; ----- Contour 7 -----
PTP {X 40.51, Y 258.85, Z 10.00, A 0, B 0, C 0}
LIN {X 40.51, Y 258.85, Z 0.00, A 0, B 0, C 0}
LIN {X 40.30, Y 258.74, Z 0.00, A 0, B 0, C 0} C_DIS
LIN {X 40.09, Y 258.64, Z 0.00, A 0, B 0, C 0} C_DIS
LIN {X 39.88, Y 258.57, Z 0.00, A 0, B 0, C 0} C_DIS
LIN {X 39.67, Y 258.50, Z 0.00, A 0, B 0, C 0} C_DIS
LIN {X 39.46, Y 258.46, Z 0.00, A 0, B 0, C 0} C_DIS
LIN {X 39.25, Y 258.42, Z 0.00, A 0, B 0, C 0} C_DIS
LIN {X 39.03, Y 258.40, Z 0.00, A 0, B 0, C 0} C_DIS
LIN {X 38.81, Y 258.38, Z 0.00, A 0, B 0, C 0} C_DIS
LIN {X 38.60, Y 258.38, Z 0.00, A 0, B 0, C 0} C_DIS
LIN {X 38.38, Y 258.38, Z 0.00, A 0, B 0, C 0} C_DIS
LIN {X 38.16, Y 258.38, Z 0.00, A 0, B 0, C 0} C_DIS
LIN {X 37.94, Y 258.39, Z 0.00, A 0, B 0, C 0} C_DIS
LIN {X 37.72, Y 258.39, Z 0.00, A 0, B 0, C 0} C_DIS
LIN {X 37.51, Y 258.40, Z 0.00, A 0, B 0, C 0} C_DIS
LIN {X 37.29, Y 258.41, Z 0.00, A 0, B 0, C 0} C_DIS
LIN {X 37.07, Y 258.41, Z 0.00, A 0, B 0, C 0} C_DIS
LIN {X 36.85, Y 258.42, Z 0.00, A 0, B 0, C 0} C_DIS
LIN {X 36.63, Y 258.42, Z 0.00, A 0, B 0, C 0} C_DIS
LIN {X 36.42, Y 258.42, Z 0.00, A 0, B 0, C 0} C_DIS
LIN {X 36.20, Y 258.42, Z 0.00, A 0, B 0, C 0} C_DIS
LIN {X 35.98, Y 258.42, Z 0.00, A 0, B 0, C 0} C_DIS
LIN {X 35.76, Y 258.42, Z 0.00, A 0, B 0, C 0} C_DIS
LIN {X 35.55, Y 258.42, Z 0.00, A 0, B 0, C 0} C_DIS
LIN {X 35.33, Y 258.42, Z 0.00, A 0, B 0, C 0} C_DIS
LIN {X 35.11, Y 258.41, Z 0.00, A 0, B 0, C 0} C_DIS
LIN {X 34.90, Y 258.41, Z 0.00, A 0, B 0, C 0} C_DIS
LIN {X 34.68, Y 258.41, Z 0.00, A 0, B 0, C 0} C_DIS
LIN {X 34.46, Y 258.41, Z 0.00, A 0, B 0, C 0} C_DIS
LIN {X 34.24, Y 258.41, Z 0.00, A 0, B 0, C 0} C_DIS
LIN {X 34.03, Y 258.40, Z 0.00, A 0, B 0, C 0} C_DIS
LIN {X 33.81, Y 258.40, Z 0.00, A 0, B 0, C 0} C_DIS
LIN {X 33.59, Y 258.40, Z 0.00, A 0, B 0, C 0} C_DIS
LIN {X 33.37, Y 258.40, Z 0.00, A 0, B 0, C 0} C_DIS
LIN {X 33.16, Y 258.40, Z 0.00, A 0, B 0, C 0} C_DIS
LIN {X 32.94, Y 258.40, Z 0.00, A 0, B 0, C 0} C_DIS
LIN {X 32.72, Y 258.40, Z 0.00, A 0, B 0, C 0} C_DIS
LIN {X 32.51, Y 258.40, Z 0.00, A 0, B 0, C 0} C_DIS
LIN {X 32.29, Y 258.40, Z 0.00, A 0, B 0, C 0} C_DIS
LIN {X 32.07, Y 258.40, Z 0.00, A 0, B 0, C 0} C_DIS
LIN {X 31.85, Y 258.40, Z 0.00, A 0, B 0, C 0} C_DIS
LIN {X 31.64, Y 258.40, Z 0.00, A 0, B 0, C 0} C_DIS
LIN {X 31.42, Y 258.40, Z 0.00, A 0, B 0, C 0} C_DIS
LIN {X 31.20, Y 258.40, Z 0.00, A 0, B 0, C 0} C_DIS
LIN {X 30.98, Y 258.40, Z 0.00, A 0, B 0, C 0} C_DIS
LIN {X 30.77, Y 258.40, Z 0.00, A 0, B 0, C 0} C_DIS
LIN {X 30.55, Y 258.40, Z 0.00, A 0, B 0, C 0} C_DIS
LIN {X 30.33, Y 258.40, Z 0.00, A 0, B 0, C 0} C_DIS
LIN {X 30.11, Y 258.41, Z 0.00, A 0, B 0, C 0} C_DIS
LIN {X 29.90, Y 258.41, Z 0.00, A 0, B 0, C 0} C_DIS
LIN {X 29.68, Y 258.41, Z 0.00, A 0, B 0, C 0} C_DIS
LIN {X 29.46, Y 258.41, Z 0.00, A 0, B 0, C 0} C_DIS
LIN {X 29.25, Y 258.41, Z 0.00, A 0, B 0, C 0} C_DIS
LIN {X 29.03, Y 258.41, Z 0.00, A 0, B 0, C 0} C_DIS
LIN {X 28.81, Y 258.41, Z 0.00, A 0, B 0, C 0} C_DIS
LIN {X 28.59, Y 258.41, Z 0.00, A 0, B 0, C 0} C_DIS
LIN {X 28.38, Y 258.41, Z 0.00, A 0, B 0, C 0} C_DIS
LIN {X 28.16, Y 258.41, Z 0.00, A 0, B 0, C 0} C_DIS
LIN {X 27.94, Y 258.41, Z 0.00, A 0, B 0, C 0} C_DIS
LIN {X 27.72, Y 258.41, Z 0.00, A 0, B 0, C 0} C_DIS
LIN {X 27.51, Y 258.41, Z 0.00, A 0, B 0, C 0} C_DIS
LIN {X 27.29, Y 258.41, Z 0.00, A 0, B 0, C 0} C_DIS
LIN {X 27.07, Y 258.41, Z 0.00, A 0, B 0, C 0} C_DIS
LIN {X 26.85, Y 258.41, Z 0.00, A 0, B 0, C 0} C_DIS
LIN {X 26.64, Y 258.41, Z 0.00, A 0, B 0, C 0} C_DIS
LIN {X 26.42, Y 258.41, Z 0.00, A 0, B 0, C 0} C_DIS
LIN {X 26.20, Y 258.41, Z 0.00, A 0, B 0, C 0} C_DIS
LIN {X 25.98, Y 258.41, Z 0.00, A 0, B 0, C 0} C_DIS
LIN {X 25.77, Y 258.41, Z 0.00, A 0, B 0, C 0} C_DIS
LIN {X 25.55, Y 258.41, Z 0.00, A 0, B 0, C 0} C_DIS
LIN {X 25.33, Y 258.41, Z 0.00, A 0, B 0, C 0} C_DIS
LIN {X 25.11, Y 258.41, Z 0.00, A 0, B 0, C 0} C_DIS
LIN {X 24.90, Y 258.41, Z 0.00, A 0, B 0, C 0} C_DIS
LIN {X 24.68, Y 258.41, Z 0.00, A 0, B 0, C 0} C_DIS
LIN {X 24.46, Y 258.41, Z 0.00, A 0, B 0, C 0} C_DIS
LIN {X 24.24, Y 258.41, Z 0.00, A 0, B 0, C 0} C_DIS
LIN {X 24.03, Y 258.41, Z 0.00, A 0, B 0, C 0} C_DIS
LIN {X 23.81, Y 258.41, Z 0.00, A 0, B 0, C 0} C_DIS
LIN {X 23.59, Y 258.41, Z 0.00, A 0, B 0, C 0} C_DIS
LIN {X 23.37, Y 258.41, Z 0.00, A 0, B 0, C 0} C_DIS
LIN {X 23.16, Y 258.41, Z 0.00, A 0, B 0, C 0} C_DIS
LIN {X 22.94, Y 258.41, Z 0.00, A 0, B 0, C 0} C_DIS
LIN {X 22.72, Y 258.41, Z 0.00, A 0, B 0, C 0} C_DIS
LIN {X 22.51, Y 258.41, Z 0.00, A 0, B 0, C 0} C_DIS
LIN {X 22.29, Y 258.41, Z 0.00, A 0, B 0, C 0} C_DIS
LIN {X 22.07, Y 258.41, Z 0.00, A 0, B 0, C 0} C_DIS
LIN {X 21.85, Y 258.40, Z 0.00, A 0, B 0, C 0} C_DIS
LIN {X 21.64, Y 258.40, Z 0.00, A 0, B 0, C 0} C_DIS
LIN {X 21.42, Y 258.40, Z 0.00, A 0, B 0, C 0} C_DIS
LIN {X 21.20, Y 258.40, Z 0.00, A 0, B 0, C 0} C_DIS
LIN {X 20.98, Y 258.40, Z 0.00, A 0, B 0, C 0} C_DIS
LIN {X 20.77, Y 258.40, Z 0.00, A 0, B 0, C 0} C_DIS
LIN {X 20.55, Y 258.40, Z 0.00, A 0, B 0, C 0} C_DIS
LIN {X 20.33, Y 258.40, Z 0.00, A 0, B 0, C 0} C_DIS
LIN {X 20.11, Y 258.40, Z 0.00, A 0, B 0, C 0} C_DIS
LIN {X 19.90, Y 258.40, Z 0.00, A 0, B 0, C 0} C_DIS
LIN {X 19.68, Y 258.40, Z 0.00, A 0, B 0, C 0} C_DIS
LIN {X 19.46, Y 258.40, Z 0.00, A 0, B 0, C 0} C_DIS
LIN {X 19.24, Y 258.40, Z 0.00, A 0, B 0, C 0} C_DIS
LIN {X 19.03, Y 258.40, Z 0.00, A 0, B 0, C 0} C_DIS
LIN {X 18.81, Y 258.40, Z 0.00, A 0, B 0, C 0} C_DIS
LIN {X 18.59, Y 258.40, Z 0.00, A 0, B 0, C 0} C_DIS
LIN {X 18.37, Y 258.40, Z 0.00, A 0, B 0, C 0} C_DIS
LIN {X 18.16, Y 258.40, Z 0.00, A 0, B 0, C 0} C_DIS
LIN {X 17.94, Y 258.40, Z 0.00, A 0, B 0, C 0} C_DIS
LIN {X 17.72, Y 258.40, Z 0.00, A 0, B 0, C 0} C_DIS
LIN {X 17.50, Y 258.40, Z 0.00, A 0, B 0, C 0} C_DIS
LIN {X 17.29, Y 258.40, Z 0.00, A 0, B 0, C 0} C_DIS
LIN {X 17.07, Y 258.40, Z 0.00, A 0, B 0, C 0} C_DIS
LIN {X 16.85, Y 258.40, Z 0.00, A 0, B 0, C 0} C_DIS
LIN {X 16.64, Y 258.40, Z 0.00, A 0, B 0, C 0} C_DIS
LIN {X 16.42, Y 258.40, Z 0.00, A 0, B 0, C 0} C_DIS
LIN {X 16.20, Y 258.40, Z 0.00, A 0, B 0, C 0} C_DIS
LIN {X 15.98, Y 258.40, Z 0.00, A 0, B 0, C 0} C_DIS
LIN {X 15.77, Y 258.40, Z 0.00, A 0, B 0, C 0} C_DIS
LIN {X 15.55, Y 258.40, Z 0.00, A 0, B 0, C 0} C_DIS
LIN {X 15.33, Y 258.40, Z 0.00, A 0, B 0, C 0} C_DIS
LIN {X 15.11, Y 258.40, Z 0.00, A 0, B 0, C 0} C_DIS
LIN {X 14.90, Y 258.40, Z 0.00, A 0, B 0, C 0} C_DIS
LIN {X 14.68, Y 258.40, Z 0.00, A 0, B 0, C 0} C_DIS
LIN {X 14.46, Y 258.41, Z 0.00, A 0, B 0, C 0} C_DIS
LIN {X 14.24, Y 258.41, Z 0.00, A 0, B 0, C 0} C_DIS
LIN {X 14.03, Y 258.41, Z 0.00, A 0, B 0, C 0} C_DIS
LIN {X 13.81, Y 258.41, Z 0.00, A 0, B 0, C 0} C_DIS
LIN {X 13.59, Y 258.41, Z 0.00, A 0, B 0, C 0} C_DIS
LIN {X 13.38, Y 258.41, Z 0.00, A 0, B 0, C 0} C_DIS
LIN {X 13.16, Y 258.41, Z 0.00, A 0, B 0, C 0} C_DIS
LIN {X 12.94, Y 258.41, Z 0.00, A 0, B 0, C 0} C_DIS
LIN {X 12.72, Y 258.41, Z 0.00, A 0, B 0, C 0} C_DIS
LIN {X 12.51, Y 258.41, Z 0.00, A 0, B 0, C 0} C_DIS
LIN {X 12.29, Y 258.41, Z 0.00, A 0, B 0, C 0} C_DIS
LIN {X 12.07, Y 258.42, Z 0.00, A 0, B 0, C 0} C_DIS
LIN {X 11.85, Y 258.42, Z 0.00, A 0, B 0, C 0} C_DIS
LIN {X 11.64, Y 258.42, Z 0.00, A 0, B 0, C 0} C_DIS
LIN {X 11.42, Y 258.42, Z 0.00, A 0, B 0, C 0} C_DIS
LIN {X 11.20, Y 258.42, Z 0.00, A 0, B 0, C 0} C_DIS
LIN {X 10.98, Y 258.42, Z 0.00, A 0, B 0, C 0} C_DIS
LIN {X 10.77, Y 258.42, Z 0.00, A 0, B 0, C 0} C_DIS
LIN {X 10.55, Y 258.42, Z 0.00, A 0, B 0, C 0} C_DIS
LIN {X 10.33, Y 258.42, Z 0.00, A 0, B 0, C 0} C_DIS
LIN {X 10.12, Y 258.42, Z 0.00, A 0, B 0, C 0} C_DIS
LIN {X 9.90, Y 258.42, Z 0.00, A 0, B 0, C 0} C_DIS
LIN {X 9.68, Y 258.42, Z 0.00, A 0, B 0, C 0} C_DIS
LIN {X 9.46, Y 258.42, Z 0.00, A 0, B 0, C 0} C_DIS
LIN {X 9.25, Y 258.42, Z 0.00, A 0, B 0, C 0} C_DIS
LIN {X 9.03, Y 258.42, Z 0.00, A 0, B 0, C 0} C_DIS
LIN {X 8.81, Y 258.42, Z 0.00, A 0, B 0, C 0} C_DIS
LIN {X 8.59, Y 258.42, Z 0.00, A 0, B 0, C 0} C_DIS
LIN {X 8.38, Y 258.42, Z 0.00, A 0, B 0, C 0} C_DIS
LIN {X 8.16, Y 258.42, Z 0.00, A 0, B 0, C 0} C_DIS
LIN {X 7.94, Y 258.42, Z 0.00, A 0, B 0, C 0} C_DIS
LIN {X 7.72, Y 258.42, Z 0.00, A 0, B 0, C 0} C_DIS
LIN {X 7.51, Y 258.42, Z 0.00, A 0, B 0, C 0} C_DIS
LIN {X 7.29, Y 258.42, Z 0.00, A 0, B 0, C 0} C_DIS
LIN {X 7.07, Y 258.41, Z 0.00, A 0, B 0, C 0} C_DIS
LIN {X 6.85, Y 258.41, Z 0.00, A 0, B 0, C 0} C_DIS
LIN {X 6.63, Y 258.41, Z 0.00, A 0, B 0, C 0} C_DIS
LIN {X 6.42, Y 258.41, Z 0.00, A 0, B 0, C 0} C_DIS
LIN {X 6.20, Y 258.41, Z 0.00, A 0, B 0, C 0} C_DIS
LIN {X 5.98, Y 258.40, Z 0.00, A 0, B 0, C 0} C_DIS
LIN {X 5.76, Y 258.40, Z 0.00, A 0, B 0, C 0} C_DIS
LIN {X 5.55, Y 258.40, Z 0.00, A 0, B 0, C 0} C_DIS
LIN {X 5.33, Y 258.40, Z 0.00, A 0, B 0, C 0} C_DIS
LIN {X 5.11, Y 258.39, Z 0.00, A 0, B 0, C 0} C_DIS
LIN {X 4.89, Y 258.39, Z 0.00, A 0, B 0, C 0} C_DIS
LIN {X 4.68, Y 258.39, Z 0.00, A 0, B 0, C 0} C_DIS
LIN {X 4.46, Y 258.38, Z 0.00, A 0, B 0, C 0} C_DIS
LIN {X 4.24, Y 258.38, Z 0.00, A 0, B 0, C 0} C_DIS
LIN {X 4.02, Y 258.38, Z 0.00, A 0, B 0, C 0} C_DIS
LIN {X 3.80, Y 258.37, Z 0.00, A 0, B 0, C 0} C_DIS
LIN {X 3.59, Y 258.36, Z 0.00, A 0, B 0, C 0} C_DIS
LIN {X 3.37, Y 258.35, Z 0.00, A 0, B 0, C 0} C_DIS
LIN {X 3.16, Y 258.32, Z 0.00, A 0, B 0, C 0} C_DIS
LIN {X 2.94, Y 258.29, Z 0.00, A 0, B 0, C 0} C_DIS
LIN {X 2.74, Y 258.24, Z 0.00, A 0, B 0, C 0} C_DIS
LIN {X 2.53, Y 258.18, Z 0.00, A 0, B 0, C 0} C_DIS
LIN {X 2.33, Y 258.09, Z 0.00, A 0, B 0, C 0} C_DIS
LIN {X 2.13, Y 257.99, Z 0.00, A 0, B 0, C 0} C_DIS
LIN {X 1.94, Y 257.86, Z 0.00, A 0, B 0, C 0} C_DIS
LIN {X 1.75, Y 257.71, Z 0.00, A 0, B 0, C 0} C_DIS
LIN {X 1.57, Y 257.52, Z 0.00, A 0, B 0, C 0} C_DIS
LIN {X 1.40, Y 257.31, Z 0.00, A 0, B 0, C 0} C_DIS
LIN {X 1.23, Y 257.08, Z 0.00, A 0, B 0, C 0} C_DIS
LIN {X 1.07, Y 256.83, Z 0.00, A 0, B 0, C 0} C_DIS
LIN {X 0.92, Y 256.56, Z 0.00, A 0, B 0, C 0} C_DIS
LIN {X 0.78, Y 256.30, Z 0.00, A 0, B 0, C 0} C_DIS
LIN {X 0.65, Y 256.03, Z 0.00, A 0, B 0, C 0} C_DIS
LIN {X 0.53, Y 255.76, Z 0.00, A 0, B 0, C 0} C_DIS
LIN {X 0.42, Y 255.48, Z 0.00, A 0, B 0, C 0} C_DIS
LIN {X 0.32, Y 255.20, Z 0.00, A 0, B 0, C 0} C_DIS
LIN {X 0.23, Y 254.91, Z 0.00, A 0, B 0, C 0} C_DIS
LIN {X 0.16, Y 254.61, Z 0.00, A 0, B 0, C 0} C_DIS
LIN {X 0.09, Y 254.30, Z 0.00, A 0, B 0, C 0} C_DIS
LIN {X 0.04, Y 253.99, Z 0.00, A 0, B 0, C 0} C_DIS
LIN {X -0.01, Y 253.66, Z 0.00, A 0, B 0, C 0} C_DIS
LIN {X -0.04, Y 253.34, Z 0.00, A 0, B 0, C 0} C_DIS
LIN {X -0.06, Y 253.01, Z 0.00, A 0, B 0, C 0} C_DIS
LIN {X -0.07, Y 252.68, Z 0.00, A 0, B 0, C 0} C_DIS
LIN {X -0.06, Y 252.35, Z 0.00, A 0, B 0, C 0} C_DIS
LIN {X -0.05, Y 252.02, Z 0.00, A 0, B 0, C 0} C_DIS
LIN {X -0.03, Y 251.70, Z 0.00, A 0, B 0, C 0} C_DIS
LIN {X 0.01, Y 251.37, Z 0.00, A 0, B 0, C 0} C_DIS
LIN {X 0.06, Y 251.06, Z 0.00, A 0, B 0, C 0} C_DIS
LIN {X 0.12, Y 250.74, Z 0.00, A 0, B 0, C 0} C_DIS
LIN {X 0.19, Y 250.44, Z 0.00, A 0, B 0, C 0} C_DIS
LIN {X 0.27, Y 250.14, Z 0.00, A 0, B 0, C 0} C_DIS
LIN {X 0.36, Y 249.85, Z 0.00, A 0, B 0, C 0} C_DIS
LIN {X 0.46, Y 249.56, Z 0.00, A 0, B 0, C 0} C_DIS
LIN {X 0.57, Y 249.29, Z 0.00, A 0, B 0, C 0} C_DIS
LIN {X 0.69, Y 249.02, Z 0.00, A 0, B 0, C 0} C_DIS
LIN {X 0.83, Y 248.76, Z 0.00, A 0, B 0, C 0} C_DIS
LIN {X 0.97, Y 248.51, Z 0.00, A 0, B 0, C 0} C_DIS
LIN {X 1.12, Y 248.27, Z 0.00, A 0, B 0, C 0} C_DIS
LIN {X 1.28, Y 248.04, Z 0.00, A 0, B 0, C 0} C_DIS
LIN {X 1.45, Y 247.82, Z 0.00, A 0, B 0, C 0} C_DIS
LIN {X 1.62, Y 247.62, Z 0.00, A 0, B 0, C 0} C_DIS
LIN {X 1.81, Y 247.43, Z 0.00, A 0, B 0, C 0} C_DIS
LIN {X 1.99, Y 247.27, Z 0.00, A 0, B 0, C 0} C_DIS
LIN {X 2.19, Y 247.13, Z 0.00, A 0, B 0, C 0} C_DIS
LIN {X 2.39, Y 247.02, Z 0.00, A 0, B 0, C 0} C_DIS
LIN {X 2.59, Y 246.93, Z 0.00, A 0, B 0, C 0} C_DIS
LIN {X 2.80, Y 246.87, Z 0.00, A 0, B 0, C 0} C_DIS
LIN {X 3.01, Y 246.82, Z 0.00, A 0, B 0, C 0} C_DIS
LIN {X 3.23, Y 246.79, Z 0.00, A 0, B 0, C 0} C_DIS
LIN {X 3.44, Y 246.77, Z 0.00, A 0, B 0, C 0} C_DIS
LIN {X 3.66, Y 246.75, Z 0.00, A 0, B 0, C 0} C_DIS
LIN {X 3.88, Y 246.74, Z 0.00, A 0, B 0, C 0} C_DIS
LIN {X 4.09, Y 246.73, Z 0.00, A 0, B 0, C 0} C_DIS
LIN {X 4.31, Y 246.72, Z 0.00, A 0, B 0, C 0} C_DIS
LIN {X 4.53, Y 246.72, Z 0.00, A 0, B 0, C 0} C_DIS
LIN {X 4.74, Y 246.71, Z 0.00, A 0, B 0, C 0} C_DIS
LIN {X 4.96, Y 246.71, Z 0.00, A 0, B 0, C 0} C_DIS
LIN {X 5.18, Y 246.71, Z 0.00, A 0, B 0, C 0} C_DIS
LIN {X 5.40, Y 246.71, Z 0.00, A 0, B 0, C 0} C_DIS
LIN {X 5.62, Y 246.71, Z 0.00, A 0, B 0, C 0} C_DIS
LIN {X 5.83, Y 246.72, Z 0.00, A 0, B 0, C 0} C_DIS
LIN {X 6.05, Y 246.72, Z 0.00, A 0, B 0, C 0} C_DIS
LIN {X 6.27, Y 246.72, Z 0.00, A 0, B 0, C 0} C_DIS
LIN {X 6.49, Y 246.73, Z 0.00, A 0, B 0, C 0} C_DIS
LIN {X 6.70, Y 246.73, Z 0.00, A 0, B 0, C 0} C_DIS
LIN {X 6.92, Y 246.73, Z 0.00, A 0, B 0, C 0} C_DIS
LIN {X 7.14, Y 246.74, Z 0.00, A 0, B 0, C 0} C_DIS
LIN {X 7.36, Y 246.74, Z 0.00, A 0, B 0, C 0} C_DIS
LIN {X 7.58, Y 246.74, Z 0.00, A 0, B 0, C 0} C_DIS
LIN {X 7.79, Y 246.74, Z 0.00, A 0, B 0, C 0} C_DIS
LIN {X 8.01, Y 246.74, Z 0.00, A 0, B 0, C 0} C_DIS
LIN {X 8.23, Y 246.75, Z 0.00, A 0, B 0, C 0} C_DIS
LIN {X 8.45, Y 246.75, Z 0.00, A 0, B 0, C 0} C_DIS
LIN {X 8.66, Y 246.75, Z 0.00, A 0, B 0, C 0} C_DIS
LIN {X 8.88, Y 246.75, Z 0.00, A 0, B 0, C 0} C_DIS
LIN {X 9.10, Y 246.75, Z 0.00, A 0, B 0, C 0} C_DIS
LIN {X 9.31, Y 246.75, Z 0.00, A 0, B 0, C 0} C_DIS
LIN {X 9.53, Y 246.75, Z 0.00, A 0, B 0, C 0} C_DIS
LIN {X 9.75, Y 246.75, Z 0.00, A 0, B 0, C 0} C_DIS
LIN {X 9.97, Y 246.75, Z 0.00, A 0, B 0, C 0} C_DIS
LIN {X 10.18, Y 246.75, Z 0.00, A 0, B 0, C 0} C_DIS
LIN {X 10.40, Y 246.75, Z 0.00, A 0, B 0, C 0} C_DIS
LIN {X 10.62, Y 246.75, Z 0.00, A 0, B 0, C 0} C_DIS
LIN {X 10.84, Y 246.75, Z 0.00, A 0, B 0, C 0} C_DIS
LIN {X 11.05, Y 246.75, Z 0.00, A 0, B 0, C 0} C_DIS
LIN {X 11.27, Y 246.75, Z 0.00, A 0, B 0, C 0} C_DIS
LIN {X 11.49, Y 246.75, Z 0.00, A 0, B 0, C 0} C_DIS
LIN {X 11.70, Y 246.75, Z 0.00, A 0, B 0, C 0} C_DIS
LIN {X 11.92, Y 246.75, Z 0.00, A 0, B 0, C 0} C_DIS
LIN {X 12.14, Y 246.74, Z 0.00, A 0, B 0, C 0} C_DIS
LIN {X 12.36, Y 246.74, Z 0.00, A 0, B 0, C 0} C_DIS
LIN {X 12.57, Y 246.74, Z 0.00, A 0, B 0, C 0} C_DIS
LIN {X 12.79, Y 246.74, Z 0.00, A 0, B 0, C 0} C_DIS
LIN {X 13.01, Y 246.74, Z 0.00, A 0, B 0, C 0} C_DIS
LIN {X 13.22, Y 246.74, Z 0.00, A 0, B 0, C 0} C_DIS
LIN {X 13.44, Y 246.74, Z 0.00, A 0, B 0, C 0} C_DIS
LIN {X 13.66, Y 246.74, Z 0.00, A 0, B 0, C 0} C_DIS
LIN {X 13.88, Y 246.74, Z 0.00, A 0, B 0, C 0} C_DIS
LIN {X 14.09, Y 246.74, Z 0.00, A 0, B 0, C 0} C_DIS
LIN {X 14.31, Y 246.74, Z 0.00, A 0, B 0, C 0} C_DIS
LIN {X 14.53, Y 246.74, Z 0.00, A 0, B 0, C 0} C_DIS
LIN {X 14.75, Y 246.74, Z 0.00, A 0, B 0, C 0} C_DIS
LIN {X 14.96, Y 246.74, Z 0.00, A 0, B 0, C 0} C_DIS
LIN {X 15.18, Y 246.74, Z 0.00, A 0, B 0, C 0} C_DIS
LIN {X 15.40, Y 246.74, Z 0.00, A 0, B 0, C 0} C_DIS
LIN {X 15.62, Y 246.74, Z 0.00, A 0, B 0, C 0} C_DIS
LIN {X 15.83, Y 246.74, Z 0.00, A 0, B 0, C 0} C_DIS
LIN {X 16.05, Y 246.74, Z 0.00, A 0, B 0, C 0} C_DIS
LIN {X 16.27, Y 246.74, Z 0.00, A 0, B 0, C 0} C_DIS
LIN {X 16.49, Y 246.74, Z 0.00, A 0, B 0, C 0} C_DIS
LIN {X 16.70, Y 246.74, Z 0.00, A 0, B 0, C 0} C_DIS
LIN {X 16.92, Y 246.73, Z 0.00, A 0, B 0, C 0} C_DIS
LIN {X 17.14, Y 246.73, Z 0.00, A 0, B 0, C 0} C_DIS
LIN {X 17.36, Y 246.73, Z 0.00, A 0, B 0, C 0} C_DIS
LIN {X 17.57, Y 246.73, Z 0.00, A 0, B 0, C 0} C_DIS
LIN {X 17.79, Y 246.73, Z 0.00, A 0, B 0, C 0} C_DIS
LIN {X 18.01, Y 246.73, Z 0.00, A 0, B 0, C 0} C_DIS
LIN {X 18.23, Y 246.73, Z 0.00, A 0, B 0, C 0} C_DIS
LIN {X 18.44, Y 246.73, Z 0.00, A 0, B 0, C 0} C_DIS
LIN {X 18.66, Y 246.74, Z 0.00, A 0, B 0, C 0} C_DIS
LIN {X 18.88, Y 246.74, Z 0.00, A 0, B 0, C 0} C_DIS
LIN {X 19.10, Y 246.74, Z 0.00, A 0, B 0, C 0} C_DIS
LIN {X 19.32, Y 246.74, Z 0.00, A 0, B 0, C 0} C_DIS
LIN {X 19.53, Y 246.74, Z 0.00, A 0, B 0, C 0} C_DIS
LIN {X 19.75, Y 246.74, Z 0.00, A 0, B 0, C 0} C_DIS
LIN {X 19.97, Y 246.74, Z 0.00, A 0, B 0, C 0} C_DIS
LIN {X 20.19, Y 246.74, Z 0.00, A 0, B 0, C 0} C_DIS
LIN {X 20.40, Y 246.74, Z 0.00, A 0, B 0, C 0} C_DIS
LIN {X 20.62, Y 246.74, Z 0.00, A 0, B 0, C 0} C_DIS
LIN {X 20.84, Y 246.74, Z 0.00, A 0, B 0, C 0} C_DIS
LIN {X 21.06, Y 246.74, Z 0.00, A 0, B 0, C 0} C_DIS
LIN {X 21.27, Y 246.74, Z 0.00, A 0, B 0, C 0} C_DIS
LIN {X 21.49, Y 246.74, Z 0.00, A 0, B 0, C 0} C_DIS
LIN {X 21.71, Y 246.74, Z 0.00, A 0, B 0, C 0} C_DIS
LIN {X 21.92, Y 246.74, Z 0.00, A 0, B 0, C 0} C_DIS
LIN {X 22.14, Y 246.74, Z 0.00, A 0, B 0, C 0} C_DIS
LIN {X 22.36, Y 246.74, Z 0.00, A 0, B 0, C 0} C_DIS
LIN {X 22.58, Y 246.74, Z 0.00, A 0, B 0, C 0} C_DIS
LIN {X 22.79, Y 246.74, Z 0.00, A 0, B 0, C 0} C_DIS
LIN {X 23.01, Y 246.74, Z 0.00, A 0, B 0, C 0} C_DIS
LIN {X 23.23, Y 246.74, Z 0.00, A 0, B 0, C 0} C_DIS
LIN {X 23.45, Y 246.74, Z 0.00, A 0, B 0, C 0} C_DIS
LIN {X 23.66, Y 246.74, Z 0.00, A 0, B 0, C 0} C_DIS
LIN {X 23.88, Y 246.74, Z 0.00, A 0, B 0, C 0} C_DIS
LIN {X 24.10, Y 246.74, Z 0.00, A 0, B 0, C 0} C_DIS
LIN {X 24.31, Y 246.74, Z 0.00, A 0, B 0, C 0} C_DIS
LIN {X 24.53, Y 246.74, Z 0.00, A 0, B 0, C 0} C_DIS
LIN {X 24.75, Y 246.74, Z 0.00, A 0, B 0, C 0} C_DIS
LIN {X 24.96, Y 246.74, Z 0.00, A 0, B 0, C 0} C_DIS
LIN {X 25.18, Y 246.75, Z 0.00, A 0, B 0, C 0} C_DIS
LIN {X 25.40, Y 246.75, Z 0.00, A 0, B 0, C 0} C_DIS
LIN {X 25.62, Y 246.75, Z 0.00, A 0, B 0, C 0} C_DIS
LIN {X 25.83, Y 246.75, Z 0.00, A 0, B 0, C 0} C_DIS
LIN {X 26.05, Y 246.75, Z 0.00, A 0, B 0, C 0} C_DIS
LIN {X 26.27, Y 246.75, Z 0.00, A 0, B 0, C 0} C_DIS
LIN {X 26.48, Y 246.75, Z 0.00, A 0, B 0, C 0} C_DIS
LIN {X 26.70, Y 246.75, Z 0.00, A 0, B 0, C 0} C_DIS
LIN {X 26.92, Y 246.75, Z 0.00, A 0, B 0, C 0} C_DIS
LIN {X 27.13, Y 246.75, Z 0.00, A 0, B 0, C 0} C_DIS
LIN {X 27.35, Y 246.75, Z 0.00, A 0, B 0, C 0} C_DIS
LIN {X 27.57, Y 246.75, Z 0.00, A 0, B 0, C 0} C_DIS
LIN {X 27.79, Y 246.75, Z 0.00, A 0, B 0, C 0} C_DIS
LIN {X 28.00, Y 246.75, Z 0.00, A 0, B 0, C 0} C_DIS
LIN {X 28.22, Y 246.74, Z 0.00, A 0, B 0, C 0} C_DIS
LIN {X 28.44, Y 246.74, Z 0.00, A 0, B 0, C 0} C_DIS
LIN {X 28.66, Y 246.74, Z 0.00, A 0, B 0, C 0} C_DIS
LIN {X 28.87, Y 246.74, Z 0.00, A 0, B 0, C 0} C_DIS
LIN {X 29.09, Y 246.74, Z 0.00, A 0, B 0, C 0} C_DIS
LIN {X 29.31, Y 246.74, Z 0.00, A 0, B 0, C 0} C_DIS
LIN {X 29.53, Y 246.73, Z 0.00, A 0, B 0, C 0} C_DIS
LIN {X 29.75, Y 246.73, Z 0.00, A 0, B 0, C 0} C_DIS
LIN {X 29.97, Y 246.73, Z 0.00, A 0, B 0, C 0} C_DIS
LIN {X 30.19, Y 246.73, Z 0.00, A 0, B 0, C 0} C_DIS
LIN {X 30.41, Y 246.72, Z 0.00, A 0, B 0, C 0} C_DIS
LIN {X 30.63, Y 246.72, Z 0.00, A 0, B 0, C 0} C_DIS
LIN {X 30.85, Y 246.71, Z 0.00, A 0, B 0, C 0} C_DIS
LIN {X 31.07, Y 246.71, Z 0.00, A 0, B 0, C 0} C_DIS
LIN {X 31.29, Y 246.70, Z 0.00, A 0, B 0, C 0} C_DIS
LIN {X 31.51, Y 246.70, Z 0.00, A 0, B 0, C 0} C_DIS
LIN {X 31.73, Y 246.71, Z 0.00, A 0, B 0, C 0} C_DIS
LIN {X 31.94, Y 246.73, Z 0.00, A 0, B 0, C 0} C_DIS
LIN {X 32.15, Y 246.77, Z 0.00, A 0, B 0, C 0} C_DIS
LIN {X 32.36, Y 246.83, Z 0.00, A 0, B 0, C 0} C_DIS
LIN {X 32.56, Y 246.92, Z 0.00, A 0, B 0, C 0} C_DIS
LIN {X 32.76, Y 247.04, Z 0.00, A 0, B 0, C 0} C_DIS
LIN {X 32.94, Y 247.18, Z 0.00, A 0, B 0, C 0} C_DIS
LIN {X 33.12, Y 247.35, Z 0.00, A 0, B 0, C 0} C_DIS
LIN {X 33.29, Y 247.55, Z 0.00, A 0, B 0, C 0} C_DIS
LIN {X 33.45, Y 247.76, Z 0.00, A 0, B 0, C 0} C_DIS
LIN {X 33.61, Y 247.98, Z 0.00, A 0, B 0, C 0} C_DIS
LIN {X 33.75, Y 248.22, Z 0.00, A 0, B 0, C 0} C_DIS
LIN {X 33.90, Y 248.46, Z 0.00, A 0, B 0, C 0} C_DIS
LIN {X 34.03, Y 248.72, Z 0.00, A 0, B 0, C 0} C_DIS
LIN {X 34.16, Y 248.98, Z 0.00, A 0, B 0, C 0} C_DIS
LIN {X 34.29, Y 249.24, Z 0.00, A 0, B 0, C 0} C_DIS
LIN {X 34.42, Y 249.51, Z 0.00, A 0, B 0, C 0} C_DIS
LIN {X 34.55, Y 249.78, Z 0.00, A 0, B 0, C 0} C_DIS
LIN {X 34.68, Y 250.04, Z 0.00, A 0, B 0, C 0} C_DIS
LIN {X 34.81, Y 250.31, Z 0.00, A 0, B 0, C 0} C_DIS
LIN {X 34.95, Y 250.56, Z 0.00, A 0, B 0, C 0} C_DIS
LIN {X 35.09, Y 250.82, Z 0.00, A 0, B 0, C 0} C_DIS
LIN {X 35.23, Y 251.07, Z 0.00, A 0, B 0, C 0} C_DIS
LIN {X 35.37, Y 251.31, Z 0.00, A 0, B 0, C 0} C_DIS
LIN {X 35.52, Y 251.56, Z 0.00, A 0, B 0, C 0} C_DIS
LIN {X 35.66, Y 251.79, Z 0.00, A 0, B 0, C 0} C_DIS
LIN {X 35.82, Y 252.03, Z 0.00, A 0, B 0, C 0} C_DIS
LIN {X 35.97, Y 252.26, Z 0.00, A 0, B 0, C 0} C_DIS
LIN {X 36.12, Y 252.50, Z 0.00, A 0, B 0, C 0} C_DIS
LIN {X 36.28, Y 252.72, Z 0.00, A 0, B 0, C 0} C_DIS
LIN {X 36.43, Y 252.95, Z 0.00, A 0, B 0, C 0} C_DIS
LIN {X 36.59, Y 253.18, Z 0.00, A 0, B 0, C 0} C_DIS
LIN {X 36.75, Y 253.40, Z 0.00, A 0, B 0, C 0} C_DIS
LIN {X 36.91, Y 253.63, Z 0.00, A 0, B 0, C 0} C_DIS
LIN {X 37.07, Y 253.85, Z 0.00, A 0, B 0, C 0} C_DIS
LIN {X 37.22, Y 254.07, Z 0.00, A 0, B 0, C 0} C_DIS
LIN {X 37.38, Y 254.29, Z 0.00, A 0, B 0, C 0} C_DIS
LIN {X 37.54, Y 254.52, Z 0.00, A 0, B 0, C 0} C_DIS
LIN {X 37.70, Y 254.74, Z 0.00, A 0, B 0, C 0} C_DIS
LIN {X 37.86, Y 254.97, Z 0.00, A 0, B 0, C 0} C_DIS
LIN {X 38.01, Y 255.19, Z 0.00, A 0, B 0, C 0} C_DIS
LIN {X 38.17, Y 255.41, Z 0.00, A 0, B 0, C 0} C_DIS
LIN {X 38.33, Y 255.64, Z 0.00, A 0, B 0, C 0} C_DIS
LIN {X 38.49, Y 255.86, Z 0.00, A 0, B 0, C 0} C_DIS
LIN {X 38.65, Y 256.07, Z 0.00, A 0, B 0, C 0} C_DIS
LIN {X 38.82, Y 256.28, Z 0.00, A 0, B 0, C 0} C_DIS
LIN {X 38.99, Y 256.48, Z 0.00, A 0, B 0, C 0} C_DIS
LIN {X 39.16, Y 256.68, Z 0.00, A 0, B 0, C 0} C_DIS
LIN {X 39.34, Y 256.87, Z 0.00, A 0, B 0, C 0} C_DIS
LIN {X 39.53, Y 257.05, Z 0.00, A 0, B 0, C 0} C_DIS
LIN {X 39.72, Y 257.22, Z 0.00, A 0, B 0, C 0} C_DIS
LIN {X 39.91, Y 257.39, Z 0.00, A 0, B 0, C 0} C_DIS
LIN {X 40.09, Y 257.56, Z 0.00, A 0, B 0, C 0} C_DIS
LIN {X 40.26, Y 257.76, Z 0.00, A 0, B 0, C 0} C_DIS
LIN {X 40.41, Y 257.97, Z 0.00, A 0, B 0, C 0} C_DIS
LIN {X 40.55, Y 258.21, Z 0.00, A 0, B 0, C 0} C_DIS
LIN {X 40.65, Y 258.49, Z 0.00, A 0, B 0, C 0} C_DIS
LIN {X 40.72, Y 258.82, Z 0.00, A 0, B 0, C 0} C_DIS
LIN {X 40.72, Y 258.82, Z 10.00, A 0, B 0, C 0}

; ----- Contour 8 -----
PTP {X 35.80, Y 257.38, Z 10.00, A 0, B 0, C 0}
LIN {X 35.80, Y 257.38, Z 0.00, A 0, B 0, C 0}
LIN {X 36.01, Y 257.23, Z 0.00, A 0, B 0, C 0} C_DIS
LIN {X 36.20, Y 257.03, Z 0.00, A 0, B 0, C 0} C_DIS
LIN {X 36.36, Y 256.79, Z 0.00, A 0, B 0, C 0} C_DIS
LIN {X 36.49, Y 256.53, Z 0.00, A 0, B 0, C 0} C_DIS
LIN {X 36.59, Y 256.24, Z 0.00, A 0, B 0, C 0} C_DIS
LIN {X 36.66, Y 255.95, Z 0.00, A 0, B 0, C 0} C_DIS
LIN {X 36.69, Y 255.64, Z 0.00, A 0, B 0, C 0} C_DIS
LIN {X 36.69, Y 255.34, Z 0.00, A 0, B 0, C 0} C_DIS
LIN {X 36.64, Y 255.05, Z 0.00, A 0, B 0, C 0} C_DIS
LIN {X 36.56, Y 254.77, Z 0.00, A 0, B 0, C 0} C_DIS
LIN {X 36.45, Y 254.49, Z 0.00, A 0, B 0, C 0} C_DIS
LIN {X 36.32, Y 254.23, Z 0.00, A 0, B 0, C 0} C_DIS
LIN {X 36.17, Y 253.97, Z 0.00, A 0, B 0, C 0} C_DIS
LIN {X 36.03, Y 253.71, Z 0.00, A 0, B 0, C 0} C_DIS
LIN {X 35.89, Y 253.46, Z 0.00, A 0, B 0, C 0} C_DIS
LIN {X 35.75, Y 253.21, Z 0.00, A 0, B 0, C 0} C_DIS
LIN {X 35.60, Y 252.96, Z 0.00, A 0, B 0, C 0} C_DIS
LIN {X 35.45, Y 252.72, Z 0.00, A 0, B 0, C 0} C_DIS
LIN {X 35.31, Y 252.49, Z 0.00, A 0, B 0, C 0} C_DIS
LIN {X 35.16, Y 252.26, Z 0.00, A 0, B 0, C 0} C_DIS
LIN {X 35.01, Y 252.02, Z 0.00, A 0, B 0, C 0} C_DIS
LIN {X 34.87, Y 251.79, Z 0.00, A 0, B 0, C 0} C_DIS
LIN {X 34.73, Y 251.55, Z 0.00, A 0, B 0, C 0} C_DIS
LIN {X 34.59, Y 251.31, Z 0.00, A 0, B 0, C 0} C_DIS
LIN {X 34.45, Y 251.06, Z 0.00, A 0, B 0, C 0} C_DIS
LIN {X 34.32, Y 250.79, Z 0.00, A 0, B 0, C 0} C_DIS
LIN {X 34.20, Y 250.52, Z 0.00, A 0, B 0, C 0} C_DIS
LIN {X 34.07, Y 250.24, Z 0.00, A 0, B 0, C 0} C_DIS
LIN {X 33.95, Y 249.96, Z 0.00, A 0, B 0, C 0} C_DIS
LIN {X 33.82, Y 249.68, Z 0.00, A 0, B 0, C 0} C_DIS
LIN {X 33.69, Y 249.41, Z 0.00, A 0, B 0, C 0} C_DIS
LIN {X 33.56, Y 249.14, Z 0.00, A 0, B 0, C 0} C_DIS
LIN {X 33.42, Y 248.89, Z 0.00, A 0, B 0, C 0} C_DIS
LIN {X 33.27, Y 248.66, Z 0.00, A 0, B 0, C 0} C_DIS
LIN {X 33.12, Y 248.44, Z 0.00, A 0, B 0, C 0} C_DIS
LIN {X 32.95, Y 248.25, Z 0.00, A 0, B 0, C 0} C_DIS
LIN {X 32.77, Y 248.09, Z 0.00, A 0, B 0, C 0} C_DIS
LIN {X 32.58, Y 247.94, Z 0.00, A 0, B 0, C 0} C_DIS
LIN {X 32.39, Y 247.81, Z 0.00, A 0, B 0, C 0} C_DIS
LIN {X 32.19, Y 247.69, Z 0.00, A 0, B 0, C 0} C_DIS
LIN {X 31.99, Y 247.59, Z 0.00, A 0, B 0, C 0} C_DIS
LIN {X 31.78, Y 247.51, Z 0.00, A 0, B 0, C 0} C_DIS
LIN {X 31.57, Y 247.44, Z 0.00, A 0, B 0, C 0} C_DIS
LIN {X 31.35, Y 247.38, Z 0.00, A 0, B 0, C 0} C_DIS
LIN {X 31.13, Y 247.33, Z 0.00, A 0, B 0, C 0} C_DIS
LIN {X 30.92, Y 247.29, Z 0.00, A 0, B 0, C 0} C_DIS
LIN {X 30.70, Y 247.26, Z 0.00, A 0, B 0, C 0} C_DIS
LIN {X 30.48, Y 247.24, Z 0.00, A 0, B 0, C 0} C_DIS
LIN {X 30.27, Y 247.22, Z 0.00, A 0, B 0, C 0} C_DIS
LIN {X 30.05, Y 247.21, Z 0.00, A 0, B 0, C 0} C_DIS
LIN {X 29.83, Y 247.21, Z 0.00, A 0, B 0, C 0} C_DIS
LIN {X 29.62, Y 247.21, Z 0.00, A 0, B 0, C 0} C_DIS
LIN {X 29.40, Y 247.21, Z 0.00, A 0, B 0, C 0} C_DIS
LIN {X 29.18, Y 247.21, Z 0.00, A 0, B 0, C 0} C_DIS
LIN {X 28.96, Y 247.22, Z 0.00, A 0, B 0, C 0} C_DIS
LIN {X 28.75, Y 247.23, Z 0.00, A 0, B 0, C 0} C_DIS
LIN {X 28.53, Y 247.24, Z 0.00, A 0, B 0, C 0} C_DIS
LIN {X 28.31, Y 247.24, Z 0.00, A 0, B 0, C 0} C_DIS
LIN {X 28.10, Y 247.25, Z 0.00, A 0, B 0, C 0} C_DIS
LIN {X 27.88, Y 247.26, Z 0.00, A 0, B 0, C 0} C_DIS
LIN {X 27.66, Y 247.26, Z 0.00, A 0, B 0, C 0} C_DIS
LIN {X 27.44, Y 247.27, Z 0.00, A 0, B 0, C 0} C_DIS
LIN {X 27.23, Y 247.27, Z 0.00, A 0, B 0, C 0} C_DIS
LIN {X 27.01, Y 247.28, Z 0.00, A 0, B 0, C 0} C_DIS
LIN {X 26.79, Y 247.28, Z 0.00, A 0, B 0, C 0} C_DIS
LIN {X 26.58, Y 247.28, Z 0.00, A 0, B 0, C 0} C_DIS
LIN {X 26.36, Y 247.28, Z 0.00, A 0, B 0, C 0} C_DIS
LIN {X 26.14, Y 247.28, Z 0.00, A 0, B 0, C 0} C_DIS
LIN {X 25.92, Y 247.28, Z 0.00, A 0, B 0, C 0} C_DIS
LIN {X 25.71, Y 247.29, Z 0.00, A 0, B 0, C 0} C_DIS
LIN {X 25.49, Y 247.29, Z 0.00, A 0, B 0, C 0} C_DIS
LIN {X 25.27, Y 247.29, Z 0.00, A 0, B 0, C 0} C_DIS
LIN {X 25.06, Y 247.28, Z 0.00, A 0, B 0, C 0} C_DIS
LIN {X 24.84, Y 247.28, Z 0.00, A 0, B 0, C 0} C_DIS
LIN {X 24.62, Y 247.28, Z 0.00, A 0, B 0, C 0} C_DIS
LIN {X 24.40, Y 247.28, Z 0.00, A 0, B 0, C 0} C_DIS
LIN {X 24.19, Y 247.28, Z 0.00, A 0, B 0, C 0} C_DIS
LIN {X 23.97, Y 247.28, Z 0.00, A 0, B 0, C 0} C_DIS
LIN {X 23.75, Y 247.28, Z 0.00, A 0, B 0, C 0} C_DIS
LIN {X 23.54, Y 247.28, Z 0.00, A 0, B 0, C 0} C_DIS
LIN {X 23.32, Y 247.27, Z 0.00, A 0, B 0, C 0} C_DIS
LIN {X 23.10, Y 247.27, Z 0.00, A 0, B 0, C 0} C_DIS
LIN {X 22.88, Y 247.27, Z 0.00, A 0, B 0, C 0} C_DIS
LIN {X 22.67, Y 247.27, Z 0.00, A 0, B 0, C 0} C_DIS
LIN {X 22.45, Y 247.27, Z 0.00, A 0, B 0, C 0} C_DIS
LIN {X 22.23, Y 247.27, Z 0.00, A 0, B 0, C 0} C_DIS
LIN {X 22.02, Y 247.27, Z 0.00, A 0, B 0, C 0} C_DIS
LIN {X 21.80, Y 247.26, Z 0.00, A 0, B 0, C 0} C_DIS
LIN {X 21.58, Y 247.26, Z 0.00, A 0, B 0, C 0} C_DIS
LIN {X 21.36, Y 247.26, Z 0.00, A 0, B 0, C 0} C_DIS
LIN {X 21.15, Y 247.26, Z 0.00, A 0, B 0, C 0} C_DIS
LIN {X 20.93, Y 247.26, Z 0.00, A 0, B 0, C 0} C_DIS
LIN {X 20.71, Y 247.26, Z 0.00, A 0, B 0, C 0} C_DIS
LIN {X 20.50, Y 247.26, Z 0.00, A 0, B 0, C 0} C_DIS
LIN {X 20.28, Y 247.26, Z 0.00, A 0, B 0, C 0} C_DIS
LIN {X 20.06, Y 247.26, Z 0.00, A 0, B 0, C 0} C_DIS
LIN {X 19.84, Y 247.26, Z 0.00, A 0, B 0, C 0} C_DIS
LIN {X 19.63, Y 247.26, Z 0.00, A 0, B 0, C 0} C_DIS
LIN {X 19.41, Y 247.25, Z 0.00, A 0, B 0, C 0} C_DIS
LIN {X 19.19, Y 247.25, Z 0.00, A 0, B 0, C 0} C_DIS
LIN {X 18.97, Y 247.25, Z 0.00, A 0, B 0, C 0} C_DIS
LIN {X 18.76, Y 247.25, Z 0.00, A 0, B 0, C 0} C_DIS
LIN {X 18.54, Y 247.25, Z 0.00, A 0, B 0, C 0} C_DIS
LIN {X 18.32, Y 247.25, Z 0.00, A 0, B 0, C 0} C_DIS
LIN {X 18.11, Y 247.25, Z 0.00, A 0, B 0, C 0} C_DIS
LIN {X 17.89, Y 247.25, Z 0.00, A 0, B 0, C 0} C_DIS
LIN {X 17.67, Y 247.25, Z 0.00, A 0, B 0, C 0} C_DIS
LIN {X 17.45, Y 247.25, Z 0.00, A 0, B 0, C 0} C_DIS
LIN {X 17.24, Y 247.25, Z 0.00, A 0, B 0, C 0} C_DIS
LIN {X 17.02, Y 247.25, Z 0.00, A 0, B 0, C 0} C_DIS
LIN {X 16.80, Y 247.25, Z 0.00, A 0, B 0, C 0} C_DIS
LIN {X 16.59, Y 247.25, Z 0.00, A 0, B 0, C 0} C_DIS
LIN {X 16.37, Y 247.25, Z 0.00, A 0, B 0, C 0} C_DIS
LIN {X 16.15, Y 247.25, Z 0.00, A 0, B 0, C 0} C_DIS
LIN {X 15.93, Y 247.25, Z 0.00, A 0, B 0, C 0} C_DIS
LIN {X 15.72, Y 247.25, Z 0.00, A 0, B 0, C 0} C_DIS
LIN {X 15.50, Y 247.25, Z 0.00, A 0, B 0, C 0} C_DIS
LIN {X 15.28, Y 247.26, Z 0.00, A 0, B 0, C 0} C_DIS
LIN {X 15.06, Y 247.26, Z 0.00, A 0, B 0, C 0} C_DIS
LIN {X 14.85, Y 247.26, Z 0.00, A 0, B 0, C 0} C_DIS
LIN {X 14.63, Y 247.26, Z 0.00, A 0, B 0, C 0} C_DIS
LIN {X 14.41, Y 247.26, Z 0.00, A 0, B 0, C 0} C_DIS
LIN {X 14.20, Y 247.26, Z 0.00, A 0, B 0, C 0} C_DIS
LIN {X 13.98, Y 247.26, Z 0.00, A 0, B 0, C 0} C_DIS
LIN {X 13.76, Y 247.26, Z 0.00, A 0, B 0, C 0} C_DIS
LIN {X 13.55, Y 247.26, Z 0.00, A 0, B 0, C 0} C_DIS
LIN {X 13.33, Y 247.26, Z 0.00, A 0, B 0, C 0} C_DIS
LIN {X 13.11, Y 247.27, Z 0.00, A 0, B 0, C 0} C_DIS
LIN {X 12.89, Y 247.27, Z 0.00, A 0, B 0, C 0} C_DIS
LIN {X 12.68, Y 247.27, Z 0.00, A 0, B 0, C 0} C_DIS
LIN {X 12.46, Y 247.27, Z 0.00, A 0, B 0, C 0} C_DIS
LIN {X 12.24, Y 247.27, Z 0.00, A 0, B 0, C 0} C_DIS
LIN {X 12.03, Y 247.27, Z 0.00, A 0, B 0, C 0} C_DIS
LIN {X 11.81, Y 247.28, Z 0.00, A 0, B 0, C 0} C_DIS
LIN {X 11.59, Y 247.28, Z 0.00, A 0, B 0, C 0} C_DIS
LIN {X 11.38, Y 247.28, Z 0.00, A 0, B 0, C 0} C_DIS
LIN {X 11.16, Y 247.28, Z 0.00, A 0, B 0, C 0} C_DIS
LIN {X 10.94, Y 247.28, Z 0.00, A 0, B 0, C 0} C_DIS
LIN {X 10.72, Y 247.28, Z 0.00, A 0, B 0, C 0} C_DIS
LIN {X 10.51, Y 247.29, Z 0.00, A 0, B 0, C 0} C_DIS
LIN {X 10.29, Y 247.29, Z 0.00, A 0, B 0, C 0} C_DIS
LIN {X 10.07, Y 247.29, Z 0.00, A 0, B 0, C 0} C_DIS
LIN {X 9.86, Y 247.29, Z 0.00, A 0, B 0, C 0} C_DIS
LIN {X 9.64, Y 247.29, Z 0.00, A 0, B 0, C 0} C_DIS
LIN {X 9.42, Y 247.29, Z 0.00, A 0, B 0, C 0} C_DIS
LIN {X 9.21, Y 247.29, Z 0.00, A 0, B 0, C 0} C_DIS
LIN {X 8.99, Y 247.29, Z 0.00, A 0, B 0, C 0} C_DIS
LIN {X 8.77, Y 247.28, Z 0.00, A 0, B 0, C 0} C_DIS
LIN {X 8.55, Y 247.28, Z 0.00, A 0, B 0, C 0} C_DIS
LIN {X 8.34, Y 247.28, Z 0.00, A 0, B 0, C 0} C_DIS
LIN {X 8.12, Y 247.27, Z 0.00, A 0, B 0, C 0} C_DIS
LIN {X 7.90, Y 247.27, Z 0.00, A 0, B 0, C 0} C_DIS
LIN {X 7.68, Y 247.27, Z 0.00, A 0, B 0, C 0} C_DIS
LIN {X 7.47, Y 247.26, Z 0.00, A 0, B 0, C 0} C_DIS
LIN {X 7.25, Y 247.25, Z 0.00, A 0, B 0, C 0} C_DIS
LIN {X 7.03, Y 247.25, Z 0.00, A 0, B 0, C 0} C_DIS
LIN {X 6.81, Y 247.24, Z 0.00, A 0, B 0, C 0} C_DIS
LIN {X 6.59, Y 247.23, Z 0.00, A 0, B 0, C 0} C_DIS
LIN {X 6.38, Y 247.22, Z 0.00, A 0, B 0, C 0} C_DIS
LIN {X 6.16, Y 247.21, Z 0.00, A 0, B 0, C 0} C_DIS
LIN {X 5.94, Y 247.21, Z 0.00, A 0, B 0, C 0} C_DIS
LIN {X 5.72, Y 247.20, Z 0.00, A 0, B 0, C 0} C_DIS
LIN {X 5.50, Y 247.20, Z 0.00, A 0, B 0, C 0} C_DIS
LIN {X 5.29, Y 247.20, Z 0.00, A 0, B 0, C 0} C_DIS
LIN {X 5.07, Y 247.21, Z 0.00, A 0, B 0, C 0} C_DIS
LIN {X 4.85, Y 247.22, Z 0.00, A 0, B 0, C 0} C_DIS
LIN {X 4.64, Y 247.24, Z 0.00, A 0, B 0, C 0} C_DIS
LIN {X 4.42, Y 247.26, Z 0.00, A 0, B 0, C 0} C_DIS
LIN {X 4.21, Y 247.29, Z 0.00, A 0, B 0, C 0} C_DIS
LIN {X 3.99, Y 247.34, Z 0.00, A 0, B 0, C 0} C_DIS
LIN {X 3.78, Y 247.39, Z 0.00, A 0, B 0, C 0} C_DIS
LIN {X 3.57, Y 247.45, Z 0.00, A 0, B 0, C 0} C_DIS
LIN {X 3.36, Y 247.53, Z 0.00, A 0, B 0, C 0} C_DIS
LIN {X 3.16, Y 247.61, Z 0.00, A 0, B 0, C 0} C_DIS
LIN {X 2.95, Y 247.71, Z 0.00, A 0, B 0, C 0} C_DIS
LIN {X 2.75, Y 247.83, Z 0.00, A 0, B 0, C 0} C_DIS
LIN {X 2.56, Y 247.96, Z 0.00, A 0, B 0, C 0} C_DIS
LIN {X 2.37, Y 248.11, Z 0.00, A 0, B 0, C 0} C_DIS
LIN {X 2.18, Y 248.27, Z 0.00, A 0, B 0, C 0} C_DIS
LIN {X 2.00, Y 248.45, Z 0.00, A 0, B 0, C 0} C_DIS
LIN {X 1.83, Y 248.65, Z 0.00, A 0, B 0, C 0} C_DIS
LIN {X 1.66, Y 248.87, Z 0.00, A 0, B 0, C 0} C_DIS
LIN {X 1.51, Y 249.10, Z 0.00, A 0, B 0, C 0} C_DIS
LIN {X 1.36, Y 249.34, Z 0.00, A 0, B 0, C 0} C_DIS
LIN {X 1.21, Y 249.60, Z 0.00, A 0, B 0, C 0} C_DIS
LIN {X 1.08, Y 249.87, Z 0.00, A 0, B 0, C 0} C_DIS
LIN {X 0.96, Y 250.14, Z 0.00, A 0, B 0, C 0} C_DIS
LIN {X 0.85, Y 250.43, Z 0.00, A 0, B 0, C 0} C_DIS
LIN {X 0.75, Y 250.73, Z 0.00, A 0, B 0, C 0} C_DIS
LIN {X 0.67, Y 251.03, Z 0.00, A 0, B 0, C 0} C_DIS
LIN {X 0.59, Y 251.33, Z 0.00, A 0, B 0, C 0} C_DIS
LIN {X 0.53, Y 251.64, Z 0.00, A 0, B 0, C 0} C_DIS
LIN {X 0.49, Y 251.96, Z 0.00, A 0, B 0, C 0} C_DIS
LIN {X 0.46, Y 252.27, Z 0.00, A 0, B 0, C 0} C_DIS
LIN {X 0.44, Y 252.59, Z 0.00, A 0, B 0, C 0} C_DIS
LIN {X 0.44, Y 252.90, Z 0.00, A 0, B 0, C 0} C_DIS
LIN {X 0.46, Y 253.22, Z 0.00, A 0, B 0, C 0} C_DIS
LIN {X 0.50, Y 253.53, Z 0.00, A 0, B 0, C 0} C_DIS
LIN {X 0.55, Y 253.84, Z 0.00, A 0, B 0, C 0} C_DIS
LIN {X 0.62, Y 254.14, Z 0.00, A 0, B 0, C 0} C_DIS
LIN {X 0.72, Y 254.43, Z 0.00, A 0, B 0, C 0} C_DIS
LIN {X 0.82, Y 254.72, Z 0.00, A 0, B 0, C 0} C_DIS
LIN {X 0.94, Y 255.00, Z 0.00, A 0, B 0, C 0} C_DIS
LIN {X 1.08, Y 255.27, Z 0.00, A 0, B 0, C 0} C_DIS
LIN {X 1.22, Y 255.54, Z 0.00, A 0, B 0, C 0} C_DIS
LIN {X 1.37, Y 255.79, Z 0.00, A 0, B 0, C 0} C_DIS
LIN {X 1.53, Y 256.03, Z 0.00, A 0, B 0, C 0} C_DIS
LIN {X 1.70, Y 256.26, Z 0.00, A 0, B 0, C 0} C_DIS
LIN {X 1.87, Y 256.47, Z 0.00, A 0, B 0, C 0} C_DIS
LIN {X 2.04, Y 256.67, Z 0.00, A 0, B 0, C 0} C_DIS
LIN {X 2.22, Y 256.86, Z 0.00, A 0, B 0, C 0} C_DIS
LIN {X 2.40, Y 257.04, Z 0.00, A 0, B 0, C 0} C_DIS
LIN {X 2.58, Y 257.19, Z 0.00, A 0, B 0, C 0} C_DIS
LIN {X 2.77, Y 257.34, Z 0.00, A 0, B 0, C 0} C_DIS
LIN {X 2.96, Y 257.46, Z 0.00, A 0, B 0, C 0} C_DIS
LIN {X 3.16, Y 257.58, Z 0.00, A 0, B 0, C 0} C_DIS
LIN {X 3.36, Y 257.67, Z 0.00, A 0, B 0, C 0} C_DIS
LIN {X 3.56, Y 257.75, Z 0.00, A 0, B 0, C 0} C_DIS
LIN {X 3.77, Y 257.81, Z 0.00, A 0, B 0, C 0} C_DIS
LIN {X 3.98, Y 257.86, Z 0.00, A 0, B 0, C 0} C_DIS
LIN {X 4.19, Y 257.89, Z 0.00, A 0, B 0, C 0} C_DIS
LIN {X 4.41, Y 257.92, Z 0.00, A 0, B 0, C 0} C_DIS
LIN {X 4.63, Y 257.93, Z 0.00, A 0, B 0, C 0} C_DIS
LIN {X 4.85, Y 257.93, Z 0.00, A 0, B 0, C 0} C_DIS
LIN {X 5.07, Y 257.93, Z 0.00, A 0, B 0, C 0} C_DIS
LIN {X 5.29, Y 257.93, Z 0.00, A 0, B 0, C 0} C_DIS
LIN {X 5.51, Y 257.92, Z 0.00, A 0, B 0, C 0} C_DIS
LIN {X 5.73, Y 257.91, Z 0.00, A 0, B 0, C 0} C_DIS
LIN {X 5.95, Y 257.89, Z 0.00, A 0, B 0, C 0} C_DIS
LIN {X 6.17, Y 257.88, Z 0.00, A 0, B 0, C 0} C_DIS
LIN {X 6.39, Y 257.87, Z 0.00, A 0, B 0, C 0} C_DIS
LIN {X 6.61, Y 257.86, Z 0.00, A 0, B 0, C 0} C_DIS
LIN {X 6.83, Y 257.86, Z 0.00, A 0, B 0, C 0} C_DIS
LIN {X 7.05, Y 257.86, Z 0.00, A 0, B 0, C 0} C_DIS
LIN {X 7.27, Y 257.85, Z 0.00, A 0, B 0, C 0} C_DIS
LIN {X 7.48, Y 257.86, Z 0.00, A 0, B 0, C 0} C_DIS
LIN {X 7.70, Y 257.86, Z 0.00, A 0, B 0, C 0} C_DIS
LIN {X 7.92, Y 257.86, Z 0.00, A 0, B 0, C 0} C_DIS
LIN {X 8.13, Y 257.86, Z 0.00, A 0, B 0, C 0} C_DIS
LIN {X 8.35, Y 257.87, Z 0.00, A 0, B 0, C 0} C_DIS
LIN {X 8.56, Y 257.87, Z 0.00, A 0, B 0, C 0} C_DIS
LIN {X 8.78, Y 257.88, Z 0.00, A 0, B 0, C 0} C_DIS
LIN {X 8.99, Y 257.88, Z 0.00, A 0, B 0, C 0} C_DIS
LIN {X 9.21, Y 257.88, Z 0.00, A 0, B 0, C 0} C_DIS
LIN {X 9.43, Y 257.89, Z 0.00, A 0, B 0, C 0} C_DIS
LIN {X 9.64, Y 257.89, Z 0.00, A 0, B 0, C 0} C_DIS
LIN {X 9.86, Y 257.89, Z 0.00, A 0, B 0, C 0} C_DIS
LIN {X 10.08, Y 257.89, Z 0.00, A 0, B 0, C 0} C_DIS
LIN {X 10.29, Y 257.89, Z 0.00, A 0, B 0, C 0} C_DIS
LIN {X 10.51, Y 257.89, Z 0.00, A 0, B 0, C 0} C_DIS
LIN {X 10.73, Y 257.89, Z 0.00, A 0, B 0, C 0} C_DIS
LIN {X 10.94, Y 257.89, Z 0.00, A 0, B 0, C 0} C_DIS
LIN {X 11.16, Y 257.89, Z 0.00, A 0, B 0, C 0} C_DIS
LIN {X 11.38, Y 257.89, Z 0.00, A 0, B 0, C 0} C_DIS
LIN {X 11.59, Y 257.89, Z 0.00, A 0, B 0, C 0} C_DIS
LIN {X 11.81, Y 257.89, Z 0.00, A 0, B 0, C 0} C_DIS
LIN {X 12.03, Y 257.89, Z 0.00, A 0, B 0, C 0} C_DIS
LIN {X 12.25, Y 257.89, Z 0.00, A 0, B 0, C 0} C_DIS
LIN {X 12.46, Y 257.89, Z 0.00, A 0, B 0, C 0} C_DIS
LIN {X 12.68, Y 257.89, Z 0.00, A 0, B 0, C 0} C_DIS
LIN {X 12.90, Y 257.89, Z 0.00, A 0, B 0, C 0} C_DIS
LIN {X 13.12, Y 257.89, Z 0.00, A 0, B 0, C 0} C_DIS
LIN {X 13.33, Y 257.88, Z 0.00, A 0, B 0, C 0} C_DIS
LIN {X 13.55, Y 257.88, Z 0.00, A 0, B 0, C 0} C_DIS
LIN {X 13.77, Y 257.88, Z 0.00, A 0, B 0, C 0} C_DIS
LIN {X 13.99, Y 257.88, Z 0.00, A 0, B 0, C 0} C_DIS
LIN {X 14.20, Y 257.88, Z 0.00, A 0, B 0, C 0} C_DIS
LIN {X 14.42, Y 257.88, Z 0.00, A 0, B 0, C 0} C_DIS
LIN {X 14.64, Y 257.88, Z 0.00, A 0, B 0, C 0} C_DIS
LIN {X 14.86, Y 257.88, Z 0.00, A 0, B 0, C 0} C_DIS
LIN {X 15.07, Y 257.88, Z 0.00, A 0, B 0, C 0} C_DIS
LIN {X 15.29, Y 257.88, Z 0.00, A 0, B 0, C 0} C_DIS
LIN {X 15.51, Y 257.88, Z 0.00, A 0, B 0, C 0} C_DIS
LIN {X 15.73, Y 257.88, Z 0.00, A 0, B 0, C 0} C_DIS
LIN {X 15.94, Y 257.88, Z 0.00, A 0, B 0, C 0} C_DIS
LIN {X 16.16, Y 257.88, Z 0.00, A 0, B 0, C 0} C_DIS
LIN {X 16.38, Y 257.88, Z 0.00, A 0, B 0, C 0} C_DIS
LIN {X 16.60, Y 257.88, Z 0.00, A 0, B 0, C 0} C_DIS
LIN {X 16.81, Y 257.88, Z 0.00, A 0, B 0, C 0} C_DIS
LIN {X 17.03, Y 257.88, Z 0.00, A 0, B 0, C 0} C_DIS
LIN {X 17.25, Y 257.88, Z 0.00, A 0, B 0, C 0} C_DIS
LIN {X 17.46, Y 257.88, Z 0.00, A 0, B 0, C 0} C_DIS
LIN {X 17.68, Y 257.88, Z 0.00, A 0, B 0, C 0} C_DIS
LIN {X 17.90, Y 257.88, Z 0.00, A 0, B 0, C 0} C_DIS
LIN {X 18.12, Y 257.88, Z 0.00, A 0, B 0, C 0} C_DIS
LIN {X 18.33, Y 257.88, Z 0.00, A 0, B 0, C 0} C_DIS
LIN {X 18.55, Y 257.88, Z 0.00, A 0, B 0, C 0} C_DIS
LIN {X 18.77, Y 257.88, Z 0.00, A 0, B 0, C 0} C_DIS
LIN {X 18.98, Y 257.88, Z 0.00, A 0, B 0, C 0} C_DIS
LIN {X 19.20, Y 257.88, Z 0.00, A 0, B 0, C 0} C_DIS
LIN {X 19.42, Y 257.88, Z 0.00, A 0, B 0, C 0} C_DIS
LIN {X 19.63, Y 257.88, Z 0.00, A 0, B 0, C 0} C_DIS
LIN {X 19.85, Y 257.88, Z 0.00, A 0, B 0, C 0} C_DIS
LIN {X 20.07, Y 257.88, Z 0.00, A 0, B 0, C 0} C_DIS
LIN {X 20.29, Y 257.88, Z 0.00, A 0, B 0, C 0} C_DIS
LIN {X 20.50, Y 257.88, Z 0.00, A 0, B 0, C 0} C_DIS
LIN {X 20.72, Y 257.89, Z 0.00, A 0, B 0, C 0} C_DIS
LIN {X 20.94, Y 257.89, Z 0.00, A 0, B 0, C 0} C_DIS
LIN {X 21.15, Y 257.89, Z 0.00, A 0, B 0, C 0} C_DIS
LIN {X 21.37, Y 257.89, Z 0.00, A 0, B 0, C 0} C_DIS
LIN {X 21.59, Y 257.89, Z 0.00, A 0, B 0, C 0} C_DIS
LIN {X 21.81, Y 257.89, Z 0.00, A 0, B 0, C 0} C_DIS
LIN {X 22.02, Y 257.89, Z 0.00, A 0, B 0, C 0} C_DIS
LIN {X 22.24, Y 257.89, Z 0.00, A 0, B 0, C 0} C_DIS
LIN {X 22.46, Y 257.89, Z 0.00, A 0, B 0, C 0} C_DIS
LIN {X 22.67, Y 257.89, Z 0.00, A 0, B 0, C 0} C_DIS
LIN {X 22.89, Y 257.89, Z 0.00, A 0, B 0, C 0} C_DIS
LIN {X 23.11, Y 257.89, Z 0.00, A 0, B 0, C 0} C_DIS
LIN {X 23.32, Y 257.89, Z 0.00, A 0, B 0, C 0} C_DIS
LIN {X 23.54, Y 257.89, Z 0.00, A 0, B 0, C 0} C_DIS
LIN {X 23.76, Y 257.89, Z 0.00, A 0, B 0, C 0} C_DIS
LIN {X 23.98, Y 257.89, Z 0.00, A 0, B 0, C 0} C_DIS
LIN {X 24.19, Y 257.89, Z 0.00, A 0, B 0, C 0} C_DIS
LIN {X 24.41, Y 257.89, Z 0.00, A 0, B 0, C 0} C_DIS
LIN {X 24.63, Y 257.89, Z 0.00, A 0, B 0, C 0} C_DIS
LIN {X 24.84, Y 257.89, Z 0.00, A 0, B 0, C 0} C_DIS
LIN {X 25.06, Y 257.88, Z 0.00, A 0, B 0, C 0} C_DIS
LIN {X 25.28, Y 257.88, Z 0.00, A 0, B 0, C 0} C_DIS
LIN {X 25.50, Y 257.88, Z 0.00, A 0, B 0, C 0} C_DIS
LIN {X 25.71, Y 257.88, Z 0.00, A 0, B 0, C 0} C_DIS
LIN {X 25.93, Y 257.88, Z 0.00, A 0, B 0, C 0} C_DIS
LIN {X 26.15, Y 257.88, Z 0.00, A 0, B 0, C 0} C_DIS
LIN {X 26.36, Y 257.88, Z 0.00, A 0, B 0, C 0} C_DIS
LIN {X 26.58, Y 257.88, Z 0.00, A 0, B 0, C 0} C_DIS
LIN {X 26.80, Y 257.88, Z 0.00, A 0, B 0, C 0} C_DIS
LIN {X 27.02, Y 257.88, Z 0.00, A 0, B 0, C 0} C_DIS
LIN {X 27.23, Y 257.87, Z 0.00, A 0, B 0, C 0} C_DIS
LIN {X 27.45, Y 257.87, Z 0.00, A 0, B 0, C 0} C_DIS
LIN {X 27.67, Y 257.87, Z 0.00, A 0, B 0, C 0} C_DIS
LIN {X 27.89, Y 257.87, Z 0.00, A 0, B 0, C 0} C_DIS
LIN {X 28.10, Y 257.87, Z 0.00, A 0, B 0, C 0} C_DIS
LIN {X 28.32, Y 257.87, Z 0.00, A 0, B 0, C 0} C_DIS
LIN {X 28.54, Y 257.87, Z 0.00, A 0, B 0, C 0} C_DIS
LIN {X 28.75, Y 257.87, Z 0.00, A 0, B 0, C 0} C_DIS
LIN {X 28.97, Y 257.87, Z 0.00, A 0, B 0, C 0} C_DIS
LIN {X 29.19, Y 257.87, Z 0.00, A 0, B 0, C 0} C_DIS
LIN {X 29.41, Y 257.87, Z 0.00, A 0, B 0, C 0} C_DIS
LIN {X 29.62, Y 257.88, Z 0.00, A 0, B 0, C 0} C_DIS
LIN {X 29.84, Y 257.88, Z 0.00, A 0, B 0, C 0} C_DIS
LIN {X 30.06, Y 257.88, Z 0.00, A 0, B 0, C 0} C_DIS
LIN {X 30.28, Y 257.88, Z 0.00, A 0, B 0, C 0} C_DIS
LIN {X 30.49, Y 257.88, Z 0.00, A 0, B 0, C 0} C_DIS
LIN {X 30.71, Y 257.89, Z 0.00, A 0, B 0, C 0} C_DIS
LIN {X 30.93, Y 257.89, Z 0.00, A 0, B 0, C 0} C_DIS
LIN {X 31.14, Y 257.89, Z 0.00, A 0, B 0, C 0} C_DIS
LIN {X 31.36, Y 257.90, Z 0.00, A 0, B 0, C 0} C_DIS
LIN {X 31.58, Y 257.90, Z 0.00, A 0, B 0, C 0} C_DIS
LIN {X 31.80, Y 257.90, Z 0.00, A 0, B 0, C 0} C_DIS
LIN {X 32.01, Y 257.90, Z 0.00, A 0, B 0, C 0} C_DIS
LIN {X 32.23, Y 257.91, Z 0.00, A 0, B 0, C 0} C_DIS
LIN {X 32.45, Y 257.91, Z 0.00, A 0, B 0, C 0} C_DIS
LIN {X 32.66, Y 257.91, Z 0.00, A 0, B 0, C 0} C_DIS
LIN {X 32.88, Y 257.90, Z 0.00, A 0, B 0, C 0} C_DIS
LIN {X 33.10, Y 257.90, Z 0.00, A 0, B 0, C 0} C_DIS
LIN {X 33.31, Y 257.89, Z 0.00, A 0, B 0, C 0} C_DIS
LIN {X 33.53, Y 257.89, Z 0.00, A 0, B 0, C 0} C_DIS
LIN {X 33.75, Y 257.88, Z 0.00, A 0, B 0, C 0} C_DIS
LIN {X 33.96, Y 257.86, Z 0.00, A 0, B 0, C 0} C_DIS
LIN {X 34.18, Y 257.85, Z 0.00, A 0, B 0, C 0} C_DIS
LIN {X 34.40, Y 257.83, Z 0.00, A 0, B 0, C 0} C_DIS
LIN {X 34.61, Y 257.81, Z 0.00, A 0, B 0, C 0} C_DIS
LIN {X 34.83, Y 257.79, Z 0.00, A 0, B 0, C 0} C_DIS
LIN {X 35.05, Y 257.76, Z 0.00, A 0, B 0, C 0} C_DIS
LIN {X 35.26, Y 257.73, Z 0.00, A 0, B 0, C 0} C_DIS
LIN {X 35.48, Y 257.70, Z 0.00, A 0, B 0, C 0} C_DIS
LIN {X 35.48, Y 257.70, Z 10.00, A 0, B 0, C 0}

PTP p_home
END
